// TwinCAT 3 PLC project Untitled2
// ProgramVersion: 3.1.4023.0
// libraries:
//   Tc2_Standard, * (Beckhoff Automation GmbH)
//   Tc2_System, * (Beckhoff Automation GmbH)
//   Tc2_Utilities, * (Beckhoff Automation GmbH)
//   Tc3_Module, * (Beckhoff Automation GmbH)
// project tree:
//   DUTs/Buffer/ E_BufferInitState.TcDUT, E_BufferState.TcDUT
//   / PlcTask.TcTTO
//   POUs/Buffer/ FB_Buffer.TcPOU
//   POUs/ MAIN.TcPOU
// (motion and I/O tree: see PLC project untitled1)
// real-time tasks:
//   TASK PlcTask: cycle T#10ms, priority 20, ADS port 350
//   TASK PlcTask1: cycle T#10ms, priority 21, ADS port 351

CONFIGURATION Untitled2
    RESOURCE PLC ON TwinCAT3
        TASK PlcTask(INTERVAL := T#10ms, PRIORITY := 21);
        PROGRAM MAIN WITH PlcTask : MAIN;
    END_RESOURCE
END_CONFIGURATION

// ---- DUTs/Buffer/E_BufferInitState.TcDUT
{attribute 'strict'}
TYPE E_BufferInitState :
(
	BUFFER_INIT_ := 0
);
END_TYPE

// ---- DUTs/Buffer/E_BufferState.TcDUT
{attribute 'strict'}
TYPE E_BufferState :
(
	BUFFER_UNINITIALIZED	:= 0,	(* Not ready to work *)
	BUFFER_INITIALIZING		:= 10,	(* Preparing to work *)
	BUFFER_READY			:= 20,	(* Ready to work, waiting for logs in buffer *)
	BUFFER_IDLE				:= 30,	(* Ready to work, waiting for logs in buffer *)
	BUFFER_ADD				:= 40,	(* Add new data to buffer base on FIFO*)
	BUFFER_GET				:= 50,	(* Get the oldest data from buffer base on FIFO*)
	BUFFER_REMOVE			:= 60,	(* Remove the oldest data from buffer base on FIFO*)
	BUFFER_RESET			:= 70	(* Remove all data of the buffer *)
);
END_TYPE

// ---- POUs/MAIN.TcPOU
PROGRAM MAIN
VAR
END_VAR

END_PROGRAM

// ---- POUs/Buffer/FB_Buffer.TcPOU
(* 
:Description: This function block allows to log the data to the buffer
*)
FUNCTION_BLOCK FB_Buffer
VAR
	sName 			: STRING;
	MAX_BUFFER_SIZE : UDINT;
	arrBuffer 		: ARRAY[0..MAX_BUFFER_SIZE] OF BYTE; (* Buffer memory used by FB_MemRingBuffer function block *)
	
	(* Internal status *)
	bActive 					: BOOL;						(*  *)
	bBusy						: BOOL;						(*  *)
	bError						: BOOL;						(*  *)
	iErrorID					: UDINT;					(*  *)
	
	(* Function blocks - buffer handling *)
	fbBuffer					: FB_MemRingBuffer;
	
	(* State machines *)
	eBufferState				: E_BufferState;
	eBufferInitState			: E_BufferInitState;
END_VAR

PROPERTY Active : REFERENCE TO BOOL
GET
Active REF= bActive;
END_GET
END_PROPERTY

PROPERTY Busy : REFERENCE TO BOOL
GET
Busy REF= bBusy;
END_GET
END_PROPERTY

PROPERTY Error : REFERENCE TO BOOL
GET
Error REF= bError;
END_GET
END_PROPERTY

PROPERTY ErrorID : REFERENCE TO UDINT
GET
ErrorID REF= iErrorID;
END_GET
END_PROPERTY

METHOD MR_FirstCycle : BOOL
VAR_INPUT
	sName 			: STRING;
	MAX_BUFFER_SIZE : UDINT;
	
END_VAR
THIS^.sName := sName;
THIS^.MAX_BUFFER_SIZE := MAX_BUFFER_SIZE;
END_METHOD

METHOD MR_Init : BOOL
VAR_INPUT
END_VAR
IF eBufferState = BUFFER_UNINITIALIZED THEN
	bBusy := TRUE;
	MR_Init := FALSE;
	eBufferState := BUFFER_INITIALIZING;
	
ELSIF eBufferState := BUFFER_READY THEN
	bBusy := FALSE;
	MR_Init := TRUE;
	
END_IF
END_METHOD

METHOD PROTECTED MS_Initializing
CASE eBufferInitState OF
	
END_CASE
END_METHOD

METHOD PROTECTED MS_Uninitialized
;
END_METHOD

METHOD PROTECTED StateMachine : BOOL
VAR_INPUT
END_VAR
CASE eBufferState OF
	BUFFER_UNINITIALIZED:
		MS_Uninitialized();
	
	BUFFER_INITIALIZING:
		
END_CASE
END_METHOD

END_FUNCTION_BLOCK
